PROGRAM P3_06_SP_CreateReport
VAR
	iStep					:INT;
	iError					:INT;
	tonResetError			:TON;
	trigStart				:R_TRIG;
	tonDelayStart			:TON;
	tonDelayDelete			:TON;
	
	fbReport				:FB_PythonScript;
END_VAR

ACT_CMDs();
trigStart(CLK:=GV.bSP_BatchClose);
IF tonResetError.Q THEN
	iError:=0;
END_IF

tonDelayStart(IN:=(iStep=10),PT:=T#1S);
tonDelayDelete(IN:=(iStep=999),PT:=T#1S);
CASE iStep OF
	
	0:
		IF trigStart.Q AND GV.stSP_Batch.sBatchName <> GV.sEmptyString AND NOT MAIn.bFirstCycle THEN
			iError:=0;
			iStep:=10;
		END_IF
		
	10:
		IF tonDelayStart.Q THEN
			iStep:=100;
		END_IF
		
	100:
		GV.stReport.bCreate_SPReport:=TRUE;
		IF fbReport.q_bBusy THEN
			iStep:=110;
		END_IF
	110:
		IF NOT fbReport.q_bBusy AND fbReport.q_bDone THEN
			iStep:=999;
		ELSIF fbReport.q_bError THEN
			iError:=iStep;
			iStep:=999;
		END_IF
	999:
		GV.stReport.bDelete_SPData:=TRUE;
		IF tonDelayDelete.Q THEN
			GV.stReport.bDelete_SPData:=FALSE;
			iStep:=0;
		END_IF
END_CASE

ACTION ACT_CMDs:
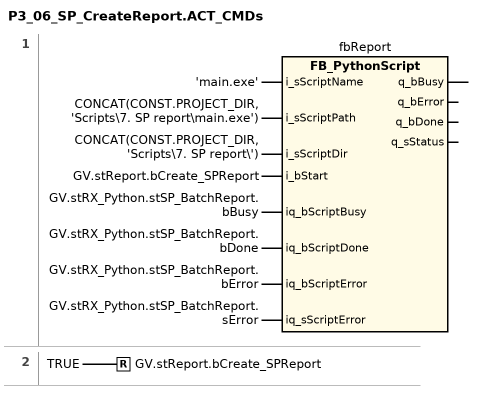
// NETWORK 1
fbReport(
    i_sScriptName := 'main.exe',
    i_sScriptPath := CONCAT(CONST.PROJECT_DIR,'Scripts\7. SP report\main.exe'),
    i_sScriptDir := CONCAT(CONST.PROJECT_DIR,'Scripts\7. SP report\'),
    i_bStart := GV.stReport.bCreate_SPReport,
    iq_bScriptBusy := GV.stRX_Python.stSP_BatchReport.bBusy,
    iq_bScriptDone := GV.stRX_Python.stSP_BatchReport.bDone,
    iq_bScriptError := GV.stRX_Python.stSP_BatchReport.bError,
    iq_sScriptError := GV.stRX_Python.stSP_BatchReport.sError); // FB_PythonScript

// NETWORK 2
GV.stReport.bCreate_SPReport R= TRUE;
END_ACTION

END_PROGRAM

(* stored: Version 1.1.0.1, ProductVersion 3.1.4024.12
   POU P3_06_SP_CreateReport: Id {e6bbc061-0a74-418f-81d3-dc946139c38f}, SpecialFunc None
   Action ACT_CMDs: Id {45f870b8-da65-420f-a80d-7fe505c7137f} *)
